// TIA Portal V16 export
// export: Created 2021-11-12T13:33:02.7448101Z, ExportSetting WithDefaults, DisplayName Totally Integrated Automation Portal, DisplayVersion V16 Update 3, DisplayName TIA Portal Version Control Interface, DisplayVersion V16 Update 2, DisplayName TIA Portal Openness, DisplayVersion V16 Update 3, DisplayName SINAMICS Startdrive Advanced, DisplayVersion V16 Update 5, DisplayName SINAMICS Startdrive G130, G150, S120, S150, SINAMICS MV, S210, DisplayVersion V16 Update 5, DisplayName SINAMICS Startdrive G110M, G120, G120C, G120D, G120P, G115D, DisplayVersion V16 Update 5, DisplayName STEP 7 Professional, DisplayVersion V16 Update 3, DisplayName STEP 7 Safety, DisplayVersion V16, DisplayName WinCC UA Professional, DisplayVersion V16 Update 3
DATA_BLOCK "STATUS_430"   // DB117
{ S7_Optimized_Access := 'TRUE' }
VERSION : 0.1
// stored: AutoNumber true, DBAccessibleFromOPCUA true, IsOnlyStoredInLoadMemory false, IsRetainMemResEnabled false, IsWriteProtectedInAS false, MemoryReserve 100
   VAR
      xxxxx___BinarySensors___xxxxx : Byte;
      "GL01-BG01" : Bool;   // Indukční snímač - Snímání kroku dopravníku
      "UC21-FC01_14" : Bool;   // 400V Dopravník ++430 OK
      xxxxx___BinaryOthers___xxxxx : Byte;
      SF02_14 : Bool;   // Conveyor Remote / Dopravník Remote
      SF02_24 : Bool;   // Conveyor Automat / Dopravník Automat
      SF03_14 : Bool;   // Conveyor Manual Backward / Dopravník Manuál Vzad
      SF03_24 : Bool;   // Conveyor Manual Forward / Dopravník Manual Vpřed
      SF04_14 : Bool;   // Conveyor Start automat / Dopravník Start automat
      SF05_12 : Bool;   // Conveyor Stop / Dopravník Stop
      xxxxx___Drives___xxxxx : Byte;
      "GL01-MA01" : Struct   // Conveyour - motor / Dopravník - motor
         Main : "UDT_Status_main";
         Specific : "UDT_Drive1_Status_specific";
         Error : "UDT_Error01";
      END_STRUCT;
      "UC21-TA01" : Struct   // Conveyour - G120 / Dopravník - měnič G120
         Main : "UDT_Status_main";
         Specific : "UDT_SINAMICS_G120_Status_specific";
         Error : "UDT_Error02";
      END_STRUCT;
      xxxxx__Alarms__xxxxx : Byte;
      ES : Struct   // E-stop
         Main { S7_SetPoint := 'True'} : "UDT_Status_main";
         Specific { S7_SetPoint := 'True'} : "UDT_DI_Mon_Status_specific";
         Error { S7_SetPoint := 'True'} : "UDT_Error01";
      END_STRUCT;
   END_VAR
BEGIN
END_DATA_BLOCK
